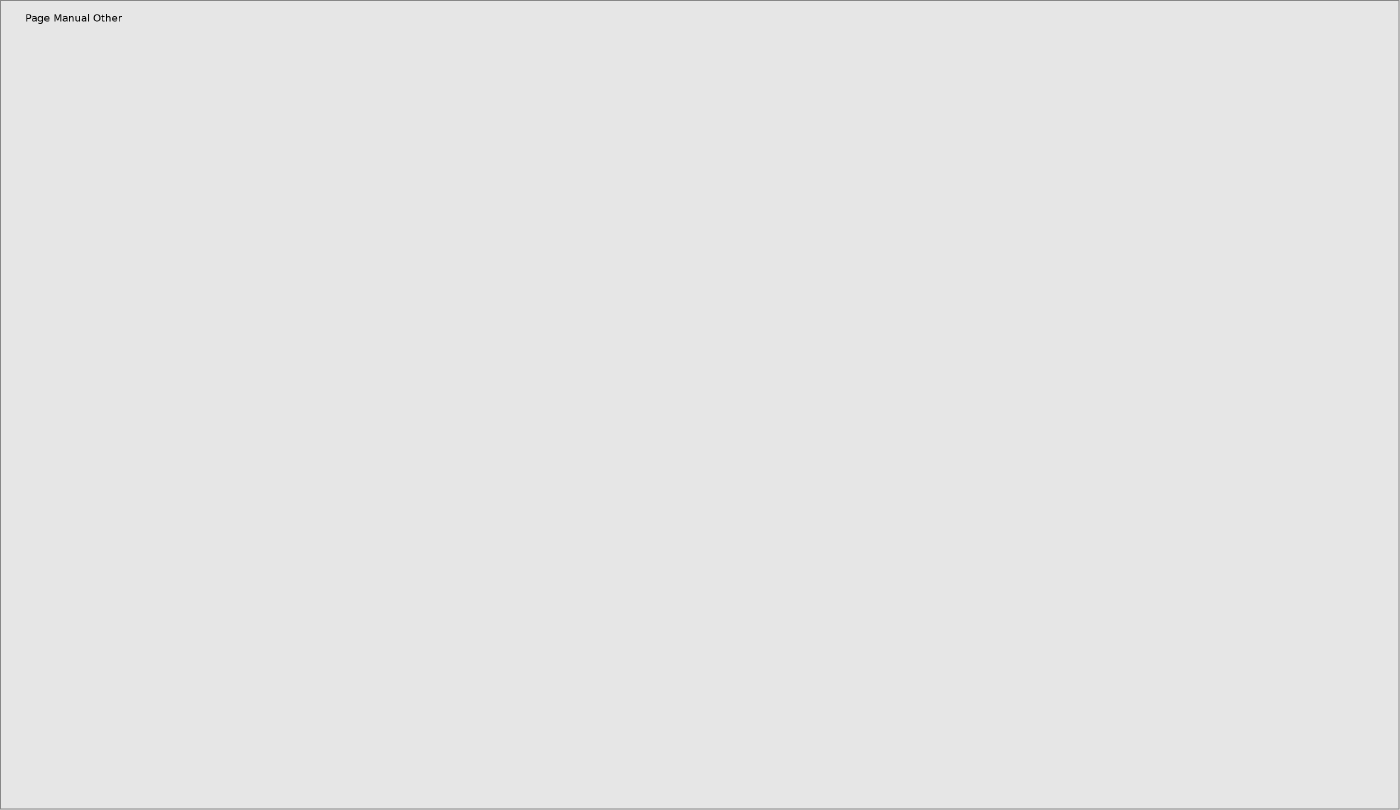
VISUALIZATION PageManualOther  // 1520x880
    Label (5,5 150x30), "Page Manual Other"
END_VISUALIZATION

(* stored: Version 1.1.0.1, ProductVersion 3.1.4024.9
   Visu PageManualOther: Id {7cfbcd7b-466e-4cbc-8466-52bf67f851ab} *)
